FUNCTION_BLOCK Test_setTestName_setsTestName EXTENDS TUnitTestBase
VAR_INPUT
END_VAR
VAR_OUTPUT
END_VAR
VAR
    UnitTest : TUnitTestUnderTest(TestSuite := 0); // not added to Test Runner
END_VAR

UnitTest.setTestName('ABCD');

Assertion.AssertEquals_STRING(
    Expected := 'ABCD.UnitTest',
    Actual   := UnitTest.TestName,
    VariableName := UnitTest.TestName);
    
TestFinished();

END_FUNCTION_BLOCK

(* stored: Version 1.1.0.1, ProductVersion 3.1.4024.4
   POU Test_setTestName_setsTestName: Id {1926a570-2039-460c-b058-b6070c6148ef}, SpecialFunc None *)
